{attribute 'GeneratedUsingTerminal: EL2521-1001-0000'}
{attribute addProperty BoxType "EL2521-1001-0000"}
{attribute addProperty Id "CtrlAT %Q*USINT1Data_OutAT %Q*UINT2"}
{attribute addProperty CRC "2422111622"}
{attribute addProperty Size "3"}
TYPE Outputs_905E7D86 :
STRUCT
	{attribute addProperty Name "Ctrl"}
	Ctrl AT %Q* : USINT;
	{attribute addProperty Name "Data_Out"}
	Data_Out AT %Q* : UINT;
END_STRUCT
END_TYPE

(* stored: Version 1.2.0.0, ProductVersion 3.1.4024.9
   DUT Outputs_905E7D86: Id {0b539f32-7adf-4e91-898e-115d200f8799} *)
